{attribute 'qualified_only'}
VAR_GLOBAL
	bStandAlone									: BOOL;		// Without superior system
	bNoPackML									: BOOL;		// Without PackML
	bGhostMode									: BOOL; 	// Without product, demo mode
	bStartCycle									: BOOL;
	bStopCycle									: BOOL;
	bServiceMode								: BOOL;
	bHoming										: BOOL;
	bReset										: BOOL;
	bChooseRecipe								: BOOL;
	bProductionEnding							: BOOL;
	bDoorOpen									: BOOL;
	
END_VAR

(* stored: Version 1.1.0.1, FileIdentifier 4508305419afe92336bef9e627c2b5b44ff1b479, FileSignature 93de5f6d654c92eb733d66f99cae4ce069dd0af71308ee5a97ebe6f18337da53fc09134cef59c459934f878aba14eed43571ef4ae79a4bf55c7ca5f1ccf165fe2f53bb0248f158b83095d3142bf39fdee360f984341717fd18d6eecf1a5623837fe49210c4f420ed7c86c7537d94d211e114271dabacfb1febfd384832b067803d39836414c19e8591bb3b6e7c0b4443b530074efb452cf9c1ba9411d1f9e5c556f54ca347a8863dd197e8ac68ba447ee86634c2e44da40b032b8400acfba53ae70ba9539f6b1db375c9f678f4c0a06b39b614aaab74cb1303ce8b2c51b8bf99444b4b58a3c0ce19461f8210a52c8aeaecd9030d692ca5d4af7220d652af8c29
   GVL GVL_StandAloneUnit: Id {527d59e3-81bf-4df9-82a4-3d2b4aa4fd7a} *)
